FUNCTION pv_float_to_dac : INT
VAR_INPUT
	pv			: LREAL;
	pv_max		: LREAL;
	pv_min		: LREAL;
	dac_max		: LREAL;
	dac_min		: LREAL;
END_VAR
VAR
END_VAR


pv_float_to_dac := LREAL_TO_INT((dac_max-dac_min)/(pv_max-pv_min)*(pv-pv_min)+dac_min);

END_FUNCTION

(* stored: Version 1.1.0.1, ProductVersion 3.1.0.36
   POU pv_float_to_dac: Id {27287405-a677-4f65-93c1-109ed01550ed}, SpecialFunc None *)
